INTERFACE I_NodeExecuteEndEvent EXTENDS I_Event

PROPERTY PUBLIC Target : I_Node
GET
END_GET
END_PROPERTY

END_INTERFACE

(* stored: Version 1.1.0.1, ProductVersion 3.1.4024.12
   Itf I_NodeExecuteEndEvent: Id {2e85dd43-4463-4c45-aae0-9bd8f223fe4e}
   Property Target: Id {ec3f884e-0ea0-43c3-96f1-19fb0f3723e1}
   Get Get: Id {6bfbe76f-3f78-46bd-8222-a68d733fb8ff} *)
